FUNCTION_BLOCK SDODatenMotor3
VAR_INPUT
END_VAR
VAR_OUTPUT
	
	Motor3Spannung: UINT;
	Motor3Strom: INT;
	Motor3Strombegrenzung: UINT;
	Motor3Regelfehler: INT;
	Motor3Geschwindigkeit: INT;
	Motor3Overloadtime: UINT;
	Motor3Overtemperature: BOOL;
	Motor3Torqueoverload: BOOL;
	Motor3Shortcirciut: BOOL;
	
END_VAR
VAR
	Motorspannung: FB_EcCoESdoRead;	
	Motorstrom: FB_EcCoESdoRead;
	Strombegrenzung: FB_EcCoESdoRead;
	Regelfehler: FB_EcCoESdoRead;
	Geschwindigkeit: FB_EcCoESdoRead;
	Overload: FB_EcCoESdoRead;
	Short_Circuit: FB_EcCoESdoRead;
	Torque_Overload: FB_EcCoESdoRead;
	Over_Temperature: FB_EcCoESdoRead;

	trigger: BOOL;
	TON_0: TON;
	TON_1: TON;
	ms: TIME;

END_VAR

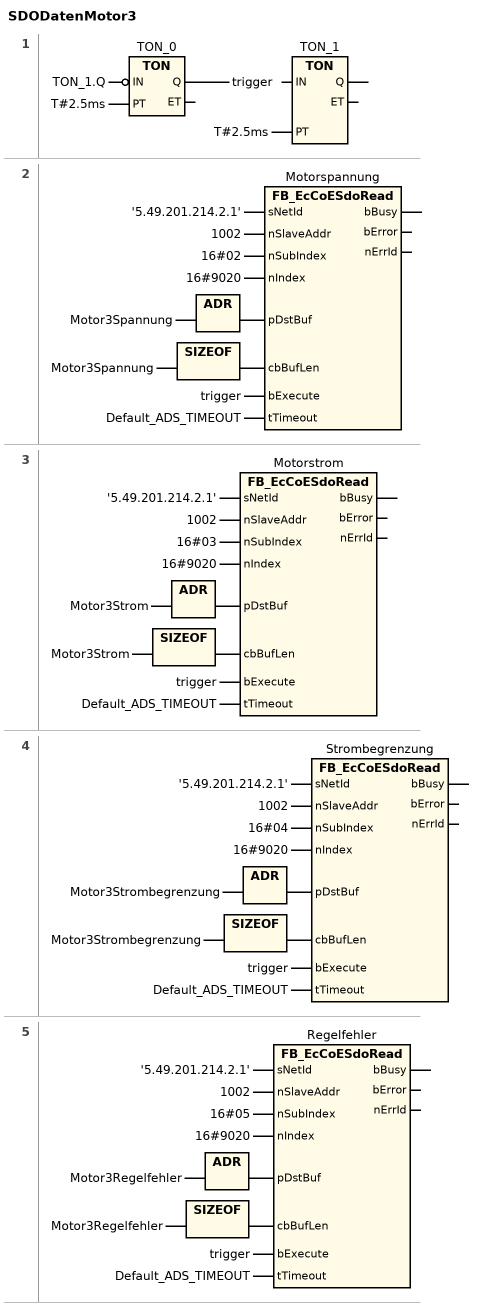
// NETWORK 1
TON_0(IN := NOT TON_1.Q, PT := T#2.5ms); // TON
trigger := TON_0.Q;
TON_1(IN := TON_0.Q, PT := T#2.5ms); // TON

// NETWORK 2
Motorspannung(
    sNetId := '5.49.201.214.2.1',
    nSlaveAddr := 1002,
    nSubIndex := 16#02,
    nIndex := 16#9020,
    pDstBuf := ADR(Motor3Spannung),
    cbBufLen := SIZEOF(Motor3Spannung),
    bExecute := trigger,
    tTimeout := Default_ADS_TIMEOUT); // FB_EcCoESdoRead

// NETWORK 3
Motorstrom(
    sNetId := '5.49.201.214.2.1',
    nSlaveAddr := 1002,
    nSubIndex := 16#03,
    nIndex := 16#9020,
    pDstBuf := ADR(Motor3Strom),
    cbBufLen := SIZEOF(Motor3Strom),
    bExecute := trigger,
    tTimeout := Default_ADS_TIMEOUT); // FB_EcCoESdoRead

// NETWORK 4
Strombegrenzung(
    sNetId := '5.49.201.214.2.1',
    nSlaveAddr := 1002,
    nSubIndex := 16#04,
    nIndex := 16#9020,
    pDstBuf := ADR(Motor3Strombegrenzung),
    cbBufLen := SIZEOF(Motor3Strombegrenzung),
    bExecute := trigger,
    tTimeout := Default_ADS_TIMEOUT); // FB_EcCoESdoRead

// NETWORK 5
Regelfehler(
    sNetId := '5.49.201.214.2.1',
    nSlaveAddr := 1002,
    nSubIndex := 16#05,
    nIndex := 16#9020,
    pDstBuf := ADR(Motor3Regelfehler),
    cbBufLen := SIZEOF(Motor3Regelfehler),
    bExecute := trigger,
    tTimeout := Default_ADS_TIMEOUT); // FB_EcCoESdoRead

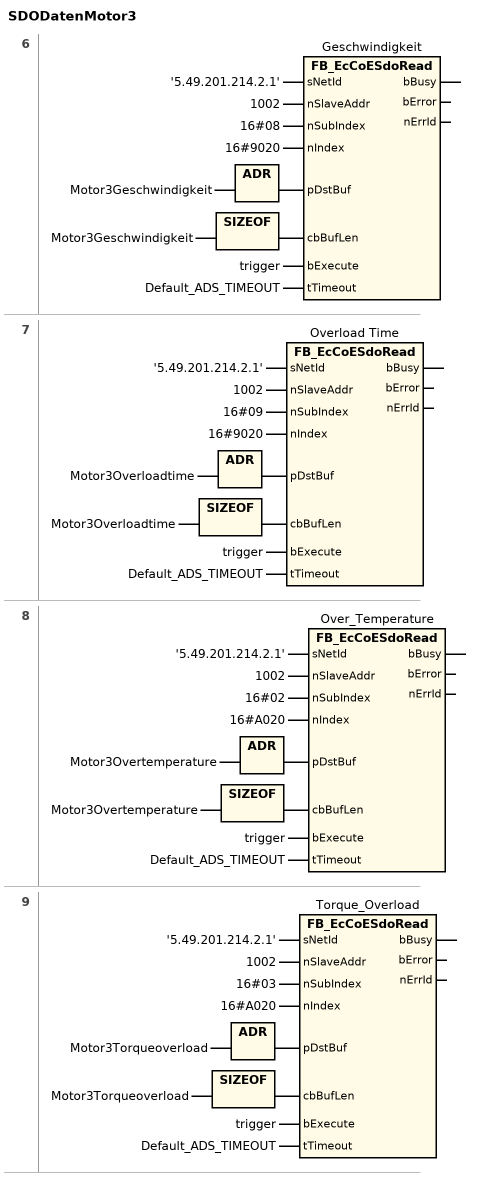
// NETWORK 6
Geschwindigkeit(
    sNetId := '5.49.201.214.2.1',
    nSlaveAddr := 1002,
    nSubIndex := 16#08,
    nIndex := 16#9020,
    pDstBuf := ADR(Motor3Geschwindigkeit),
    cbBufLen := SIZEOF(Motor3Geschwindigkeit),
    bExecute := trigger,
    tTimeout := Default_ADS_TIMEOUT); // FB_EcCoESdoRead

// NETWORK 7
Overload Time(
    sNetId := '5.49.201.214.2.1',
    nSlaveAddr := 1002,
    nSubIndex := 16#09,
    nIndex := 16#9020,
    pDstBuf := ADR(Motor3Overloadtime),
    cbBufLen := SIZEOF(Motor3Overloadtime),
    bExecute := trigger,
    tTimeout := Default_ADS_TIMEOUT); // FB_EcCoESdoRead

// NETWORK 8
Over_Temperature(
    sNetId := '5.49.201.214.2.1',
    nSlaveAddr := 1002,
    nSubIndex := 16#02,
    nIndex := 16#A020,
    pDstBuf := ADR(Motor3Overtemperature),
    cbBufLen := SIZEOF(Motor3Overtemperature),
    bExecute := trigger,
    tTimeout := Default_ADS_TIMEOUT); // FB_EcCoESdoRead

// NETWORK 9
Torque_Overload(
    sNetId := '5.49.201.214.2.1',
    nSlaveAddr := 1002,
    nSubIndex := 16#03,
    nIndex := 16#A020,
    pDstBuf := ADR(Motor3Torqueoverload),
    cbBufLen := SIZEOF(Motor3Torqueoverload),
    bExecute := trigger,
    tTimeout := Default_ADS_TIMEOUT); // FB_EcCoESdoRead

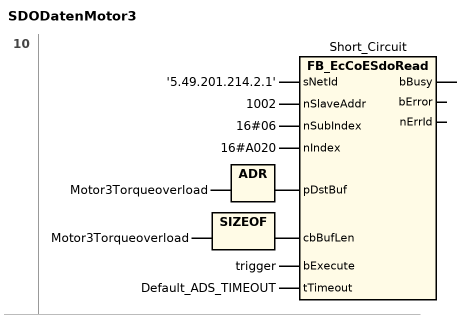
// NETWORK 10
Short_Circuit(
    sNetId := '5.49.201.214.2.1',
    nSlaveAddr := 1002,
    nSubIndex := 16#06,
    nIndex := 16#A020,
    pDstBuf := ADR(Motor3Torqueoverload),
    cbBufLen := SIZEOF(Motor3Torqueoverload),
    bExecute := trigger,
    tTimeout := Default_ADS_TIMEOUT); // FB_EcCoESdoRead

END_FUNCTION_BLOCK

(* stored: Version 1.1.0.1, ProductVersion 3.1.4022.3
   POU SDODatenMotor3: Id {5bc7d266-ec51-483d-8fad-12dbadf748de}, SpecialFunc None *)
